FUNCTION_BLOCK TransportSequenceFaultReaction EXTENDS TransportSequence IMPLEMENTS ZCore.ISequence
VAR
  _step : ZCore.Step(TransportStep.FaultReactionBegin, TransportStep.FaultReactionEnd);
  _timerSim : ZAux.Timer;
END_VAR

IF OnStart(_step) THEN
  ; // init custom sequence variables here ...
END_IF

REPEAT
  LogStep();

  CASE _step.Index OF
    (* -------------------------------------------------------------------------------------------------------------------------------- *)
    TransportStep.FaultReactionBegin:
    (* -------------------------------------------------------------------------------------------------------------------------------- *)
      IF _step.OnEntry()
      THEN
        _axis.HorizontalX.StopAsync(startToken:=THIS^);
        _axis.VerticalZ.StopAsync(startToken:=THIS^);
			END_IF
      
      Await2(obj1:=_axis.HorizontalX, obj2:=_axis.VerticalZ, nextStep:=TransportStep.FaultReactionVerticalUp);

    (* -------------------------------------------------------------------------------------------------------------------------------- *)
    TransportStep.FaultReactionVerticalUp:
    (* -------------------------------------------------------------------------------------------------------------------------------- *)
      IF _step.OnEntry()
      THEN        
        _axis.VerticalZ.MoveAbsoluteAsync(startToken:=THIS^, position:=_data.Machine.VerticalTopPos, speed:=_data.Machine.Slowspeed);
      END_IF
      
      Await(obj1:=_axis.VerticalZ, nextStep:=TransportStep.FaultReactionEnd);

    (* -------------------------------------------------------------------------------------------------------------------------------- *)
    TransportStep.FaultReactionEnd:
    (* -------------------------------------------------------------------------------------------------------------------------------- *)    
      SetBusy(FALSE);
  
  ELSE
    Abort('sequence contains unhandled step');
  END_CASE
UNTIL _step.IsNotRepeatable() OR_ELSE NOT Busy END_REPEAT

END_FUNCTION_BLOCK

(* stored: Version 1.1.0.1
   POU TransportSequenceFaultReaction: Id {f6d1f354-156c-4133-b9e8-363e7cb3361b}, SpecialFunc None *)
